(*

.. <legal notes>

legal notes
=================
| SPDX-FileCopyrightText: © 2026 Oleksandr Tiutyk <trofimich@gmail.com>
| SPDX-License-Identifier: LGPL-3.0-only
| For details check: LGPL-3.0-only_

.. _LGPL-3.0-only: https://www.gnu.org/licenses/lgpl-3.0.en.html

.. </legal notes>

*)

{attribute 'no_explicit_call' := 'do not call this function block directly'} 
FUNCTION_BLOCK AutomationRunner EXTENDS Core.Object IMPLEMENTS IAutomationRunner
VAR_OUTPUT
	InitializationErrorMessage : Core.ERROR_MESSAGE;
END_VAR
VAR
	_ClassName : STRING := __POUNAME();

	_State : AUTOMATION_RUNNER_STATE;
END_VAR
VAR_STAT
	{attribute 'hide'} 
    _InstanceCounter : BYTE := 0;
END_VAR

{attribute 'monitoring' := 'call'}
PROPERTY ClassName : STRING
GET
ClassName := _ClassName;
END_GET
END_PROPERTY

{attribute 'monitoring' := 'call'}
PROPERTY FINAL CodeExecutionPhase : BOOL
GET
CodeExecutionPhase := GlobalState.CodeExecutionPhase;
END_GET
END_PROPERTY

{attribute 'monitoring' := 'call'}
PROPERTY FINAL CycleCounter : LWORD
GET
CycleCounter := GlobalState.CycleCounter;
END_GET
END_PROPERTY

METHOD FINAL Execute
VAR_IN_OUT CONSTANT
	controllers : ARRAY [*] OF IAutomationController;
END_VAR
VAR
	i : DINT;
			
	initialized : BOOL;
END_VAR
GlobalState.CodeExecutionPhase := TRUE;

Core.SystemDateTimeManager.Execute();		

Core.LogManager.Execute();

IF Core.SystemDateTimeManager.SystemTimeValid THEN
	//_ExecutionContext.CycleLocalStartTime := Core.SystemDateTimeManager.SystemLocalDateTime;
	//_ExecutionContext.CycleUtcStartTime := Core.SystemDateTimeManager.SystemUtcDateTime;
	
	CASE _State OF
		AUTOMATION_RUNNER_STATE.INITIALIZING:
			IF UPPER_BOUND(controllers, 1) - LOWER_BOUND(controllers, 1) < 0 THEN
				_State := AUTOMATION_RUNNER_STATE.INITIALIZATION_FAILED;		
				InitializationErrorMessage := "No controllers to run";
				RETURN;		
			END_IF

			initialized := TRUE;
			
			FOR i := LOWER_BOUND(controllers, 1) TO UPPER_BOUND(controllers, 1) DO
				IF Controllers[i] = 0 THEN
					_State := AUTOMATION_RUNNER_STATE.INITIALIZATION_FAILED;
					InitializationErrorMessage := Core.WideStrings.Concat255("controller[", TO_WSTRING(i), "] is null");
					EXIT;					
				END_IF

				Controllers[i].Initialize();
				
				CASE Controllers[i].State OF
					AUTOMATION_CONTROLLER_STATE.FAULT:
						_State := AUTOMATION_RUNNER_STATE.INITIALIZATION_FAILED;
						InitializationErrorMessage := Core.WideStrings.Concat255("controller[", TO_WSTRING(i), "] failed");
						EXIT;
						
					AUTOMATION_CONTROLLER_STATE.INITIAL:
						initialized := FALSE;						
				END_CASE
			END_FOR		
			
			IF initialized THEN
				_State := AUTOMATION_RUNNER_STATE.RUNNING;
			END_IF
		
		AUTOMATION_RUNNER_STATE.RUNNING:
			FOR i := LOWER_BOUND(controllers, 1) TO UPPER_BOUND(controllers, 1) DO
				Controllers[i].Execute();			
			END_FOR		
	END_CASE

END_IF

Core.ExceptionManager.Cleanup();
Core.DynamicMemoryManager.CleanupMemory();

GlobalState.CycleCounter := GlobalState.CycleCounter + 1;
GlobalState.CodeExecutionPhase := FALSE;
END_METHOD

METHOD FB_init : BOOL
VAR_INPUT
	(* if TRUE, the retain variables are initialized (warm start / cold start)*)
	bInitRetains	: BOOL;
	(* if TRUE, the instance afterwards gets moved into the copy code (online change)*)
	bInCopyCode	: BOOL;
END_VAR
_InstanceCounter := _InstanceCounter + 1;
END_METHOD

{attribute 'monitoring' := 'call'}
PROPERTY NamespaceName : STRING
GET
NamespaceName := CurrentNamespace.Name;
END_GET
END_PROPERTY

{attribute 'monitoring' := 'call'}
PROPERTY SelfSize : ULINT
GET
SelfSize := XSIZEOF(THIS^);
END_GET
END_PROPERTY

{attribute 'monitoring' := 'call'}
PROPERTY FINAL State : AUTOMATION_RUNNER_STATE
GET
State := _State;
END_GET
END_PROPERTY

{attribute 'monitoring' := 'call'}
PROPERTY StateName : STRING
GET
StateName := TO_STRING(_State);
END_GET
END_PROPERTY

END_FUNCTION_BLOCK

(* stored: Version 1.1.0.1
   POU AutomationRunner: Id {142225ba-ead8-4c1c-a7bd-6f13f6bbc05e}, SpecialFunc None
   Property ClassName: Id {c0a74b6f-d74a-495c-97f7-b85bba3b2667}
   Get Get: Id {42ced8f1-8292-4d64-9005-f1d881faf538}
   Property CodeExecutionPhase: Id {c4f37de1-c494-4e98-bff8-e5a29ee70657}
   Get Get: Id {cca78e62-5e2b-457e-91fc-ec64208d7a39}
   Property CycleCounter: Id {b44e2d41-8633-4c1c-ad38-18becdb27866}
   Get Get: Id {3b2c949f-bedb-4db8-bff6-1b934597b8a9}
   Method Execute: Id {cddfd6b6-d698-4df7-b955-3cc076d37dea}
   Method FB_init: Id {d9dc6fd8-04ec-4586-b655-20027fb1c3eb}
   Property NamespaceName: Id {631acbbf-d63d-4152-93f4-5099a5ad032e}
   Get Get: Id {4f5331e9-77d5-4a4f-bcca-1aa45e235864}
   Property SelfSize: Id {92318db9-3f18-4ff5-a634-be283d0bf91b}
   Get Get: Id {cb1c0e7d-8133-4dbc-9b47-0a21e7b7ce5a}
   Property State: Id {f2dce25c-3e10-4ca3-baf9-9dc113064c6d}
   Get Get: Id {62ee6d12-cc93-4e49-aed3-a8cc7d8a5a22}
   Property StateName: Id {58b8e5b1-72bd-47bf-97d3-37a11efb695b}
   Get Get: Id {b78f5aab-7d64-4910-9ee4-7e1a78e3105f} *)
